{attribute 'qualified_only'}
{attribute 'strict'}
{attribute 'to_string'}
TYPE E_MESSAGE_CTRL :
(
	MSG_CTRL_NULL,
	MSG_CTRL_INIT   := 10,
  MSG_CTRL_IDLE   := 30,
  MSG_CTRL_WRITE  := 50
)UINT;
END_TYPE

(* stored: Version 1.1.0.1, ProductVersion 3.1.4026.18
   DUT E_MESSAGE_CTRL: Id {8087737e-4763-4f02-8312-755fcb6fa599} *)
